FUNCTION_BLOCK Sensor (* Composite Function Block Type *)
  (* Standard: 61499-2 *)
  (* Version 0.0, 9/14/2008, Horst Mayer, nxtControl GmbH, template *)
  PACKAGE Main;
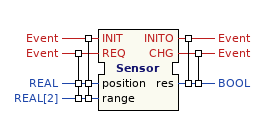
  EVENT_INPUT
    INIT WITH position, range;
    REQ WITH position, range; (* Normal Execution Request *)
  END_EVENT
  EVENT_OUTPUT
    INITO WITH res;
    CHG WITH res; (* Execution Confirmation *)
  END_EVENT
  VAR_INPUT
    position : REAL;
    range : ARRAY [0..1] OF REAL;
  END_VAR
  VAR_OUTPUT
    res : BOOL;
  END_VAR
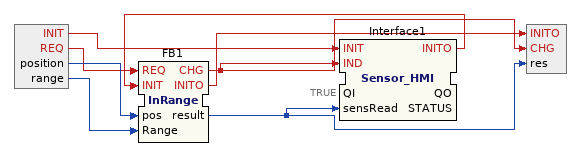
  FBS
    Interface1 : Sensor_HMI(QI := TRUE);
    FB1 : InRange;
  END_FBS
  EVENT_CONNECTIONS
    REQ TO FB1.REQ;
    FB1.CHG TO CHG;
    INIT TO Interface1.INIT;
    FB1.CHG TO Interface1.IND;
    Interface1.INITO TO FB1.INIT;
    FB1.INITO TO INITO;
  END_CONNECTIONS
  DATA_CONNECTIONS
    FB1.result TO res;
    position TO FB1.pos;
    range TO FB1.Range;
    FB1.result TO Interface1.sensRead;
  END_CONNECTIONS
END_FUNCTION_BLOCK
